Staubli VAL3: recvRosMsg.pgx

program recvRosMsg(sio& x_sSocket, Prefix& x_pPrefix, Header& x_hHeader, Body& x_bBody, num& x_nConnFlag, RosSimpleMsg& x_rMsg, bool& x_bValidFlag)
begin
  // Copyright (c) 2021, Institute for Factory Automation and Production Systems (FAPS)
  //
  // Licensed under the Apache License, Version 2.0 (the "License");
  // you may not use this file except in compliance with the License.
  // You may obtain a copy of the License at
  //
  //     http://www.apache.org/licenses/LICENSE-2.0
  //
  // Unless required by applicable law or agreed to in writing, software
  // distributed under the License is distributed on an "AS IS" BASIS,
  // WITHOUT WARRANTIES OR CONDITIONS OF ANY KIND, either express or implied.
  // See the License for the specific language governing permissions and
  // limitations under the License.


  // attempt to receive the data of the message (prefix and header are in x_msg)
  x_pPrefix.nLength=x_rMsg.prefix.nLength
  x_hHeader.nMsgType=x_rMsg.header.nMsgType
  x_hHeader.nCommType=x_rMsg.header.nCommType
  x_hHeader.nReplyCode=x_rMsg.header.nReplyCode

  call recvData(x_sSocket,x_bBody.nData,x_nConnFlag,x_bValidFlag)
end
